% RSLogix 500 project O2 Sensor Calibration.RSS, saved by version 8.30.00.16 %
PROJECT "SIM_PLC"    % processor: Bul.1763 MicroLogix 1100 Series B %

PROGRAM FILES
  LAD 2 "MAIN"  4 rungs
  LAD 3 "IO"  5 rungs
  LAD 4 "CALIBRATE"  12 rungs
  LAD 5 "GAS VALVES"  3 rungs  % O2 Concentration Values to be read by O2 Sensor %

DATA FILES
  O0 OUTPUT  5 elements
  I1 INPUT  7 elements
  S2 STATUS  66 elements
  B3 BINARY  1 elements
  T4 TIMER  4 elements
  C5 COUNTER  1 elements
  R6 CONTROL  1 elements
  N7 INTEGER  14 elements
  F8 FLOAT  5 elements

LADDER 2 "MAIN"
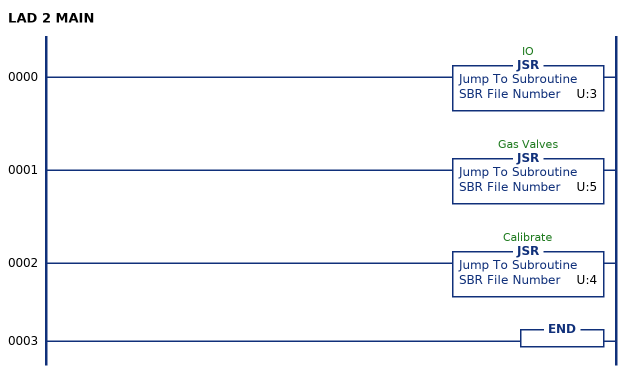
% Rung: 0 %
SOR JSR U:3 EOR
%   U:3  "IO" %
% Rung: 1 %
SOR JSR U:5 EOR
%   U:5  "Gas Valves" %
% Rung: 2 %
SOR JSR U:4 EOR
%   U:4  "Calibrate" %
% Rung: 3 %
SOR END EOR

LADDER 3 "IO"
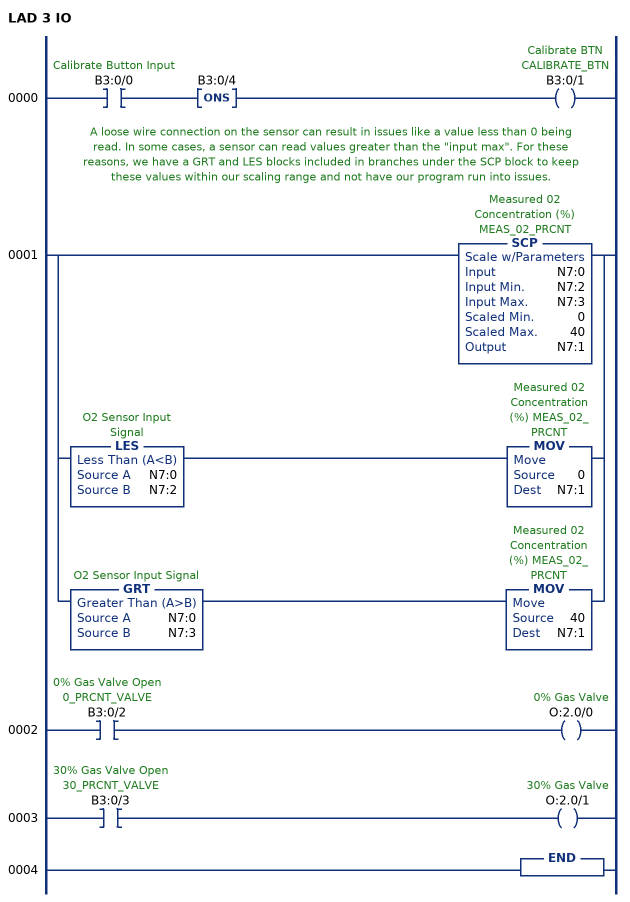
% Rung: 0 %
SOR XIC B3:0/0 ONS B3:0/4 OTE B3:0/1 EOR
%   B3:0/0  "Calibrate Button Input" %
%   B3:0/1  CALIBRATE_BTN  "Calibrate BTN" %
% Rung: 1 %
% A loose wire connection on the sensor can result in issues like a value less than 0 being read. In some cases, a sensor can read values greater than the "input max". For these reasons, we have a GRT and LES blocks included in branches under the SCP block to keep these values within our scaling range and not have our program run into issues. %
SOR BST SCP N7:0 N7:2 N7:3 0 40 N7:1 NXB LES N7:0 N7:2 MOV 0 N7:1 NXB GRT N7:0 N7:3 MOV 40 N7:1 BND EOR
%   N7:0  "O2 Sensor Input Signal" %
%   N7:2  "O2 Input Min" %
%   N7:3  "O2 Input Max" %
%   N7:1  MEAS_02_PRCNT  "Measured 02 Concentration (%)" %
% Rung: 2 %
SOR XIC B3:0/2 OTE O:2.0/0 EOR
%   B3:0/2  0_PRCNT_VALVE  "0% Gas Valve Open" %
%   O:2.0/0  "0% Gas Valve" %
% Rung: 3 %
SOR XIC B3:0/3 OTE O:2.0/1 EOR
%   B3:0/3  30_PRCNT_VALVE  "30% Gas Valve Open" %
%   O:2.0/1  "30% Gas Valve" %
% Rung: 4 %
SOR END EOR

LADDER 4 "CALIBRATE"
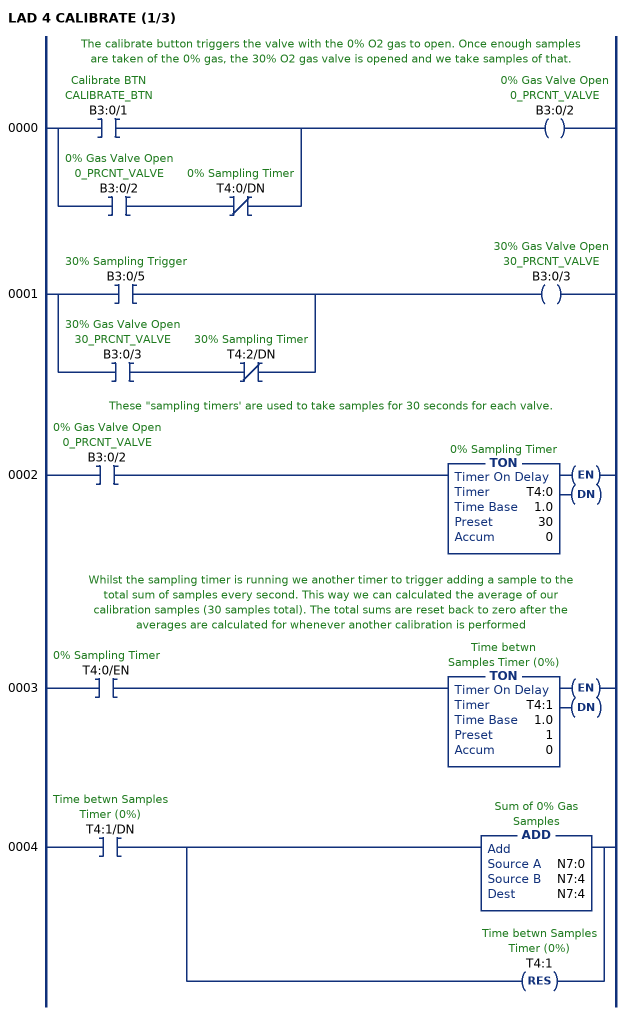
% Rung: 0 %
% The calibrate button triggers the valve with the 0% O2 gas to open. Once enough samples are taken of the 0% gas, the 30% O2 gas valve is opened and we take samples of that. %
SOR BST XIC B3:0/1 NXB XIC B3:0/2 XIO T4:0/DN BND OTE B3:0/2 EOR
%   B3:0/1  CALIBRATE_BTN  "Calibrate BTN" %
%   B3:0/2  0_PRCNT_VALVE  "0% Gas Valve Open" %
%   T4:0  "0% Sampling Timer" %
% Rung: 1 %
SOR BST XIC B3:0/5 NXB XIC B3:0/3 XIO T4:2/DN BND OTE B3:0/3 EOR
%   B3:0/5  "30% Sampling Trigger" %
%   B3:0/3  30_PRCNT_VALVE  "30% Gas Valve Open" %
%   T4:2  "30% Sampling Timer" %
% Rung: 2 %
% These "sampling timers' are used to take samples for 30 seconds for each valve. %
SOR XIC B3:0/2 TON T4:0 1.0 30 0 EOR
%   B3:0/2  0_PRCNT_VALVE  "0% Gas Valve Open" %
%   T4:0  "0% Sampling Timer" %
% Rung: 3 %
% Whilst the sampling timer is running we another timer to trigger adding a sample to the total sum of samples every second. This way we can calculated the average of our calibration samples (30 samples total). The total sums are reset back to zero after the averages are calculated for whenever another calibration is performed %
SOR XIC T4:0/EN TON T4:1 1.0 1 0 EOR
%   T4:0  "0% Sampling Timer" %
%   T4:1  "Time betwn Samples Timer (0%)" %
% Rung: 4 %
SOR XIC T4:1/DN BST ADD N7:0 N7:4 N7:4 NXB RES T4:1 BND EOR
%   T4:1  "Time betwn Samples Timer (0%)" %
%   N7:0  "O2 Sensor Input Signal" %
%   N7:4  "Sum of 0% Gas Samples" %

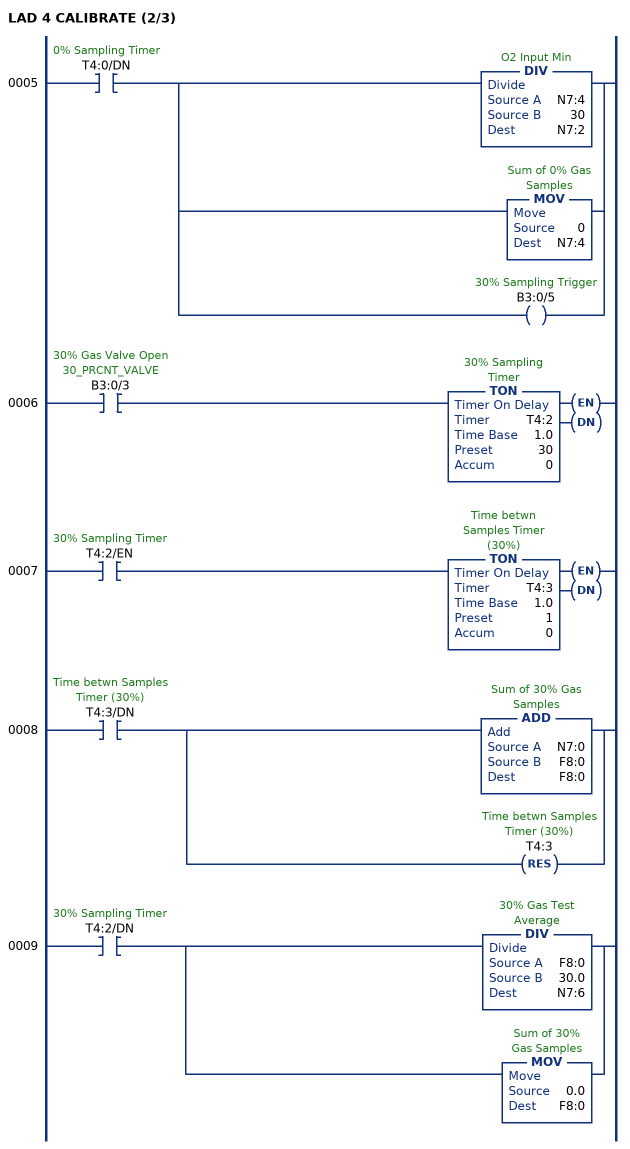
% Rung: 5 %
SOR XIC T4:0/DN BST DIV N7:4 30 N7:2 NXB MOV 0 N7:4 NXB OTE B3:0/5 BND EOR
%   T4:0  "0% Sampling Timer" %
%   N7:4  "Sum of 0% Gas Samples" %
%   N7:2  "O2 Input Min" %
%   B3:0/5  "30% Sampling Trigger" %
% Rung: 6 %
SOR XIC B3:0/3 TON T4:2 1.0 30 0 EOR
%   B3:0/3  30_PRCNT_VALVE  "30% Gas Valve Open" %
%   T4:2  "30% Sampling Timer" %
% Rung: 7 %
SOR XIC T4:2/EN TON T4:3 1.0 1 0 EOR
%   T4:2  "30% Sampling Timer" %
%   T4:3  "Time betwn Samples Timer (30%)" %
% Rung: 8 %
SOR XIC T4:3/DN BST ADD N7:0 F8:0 F8:0 NXB RES T4:3 BND EOR
%   T4:3  "Time betwn Samples Timer (30%)" %
%   N7:0  "O2 Sensor Input Signal" %
%   F8:0  "Sum of 30% Gas Samples" %
% Rung: 9 %
SOR XIC T4:2/DN BST DIV F8:0 30.0 N7:6 NXB MOV 0.0 F8:0 BND EOR
%   T4:2  "30% Sampling Timer" %
%   F8:0  "Sum of 30% Gas Samples" %
%   N7:6  "30% Gas Test Average" %

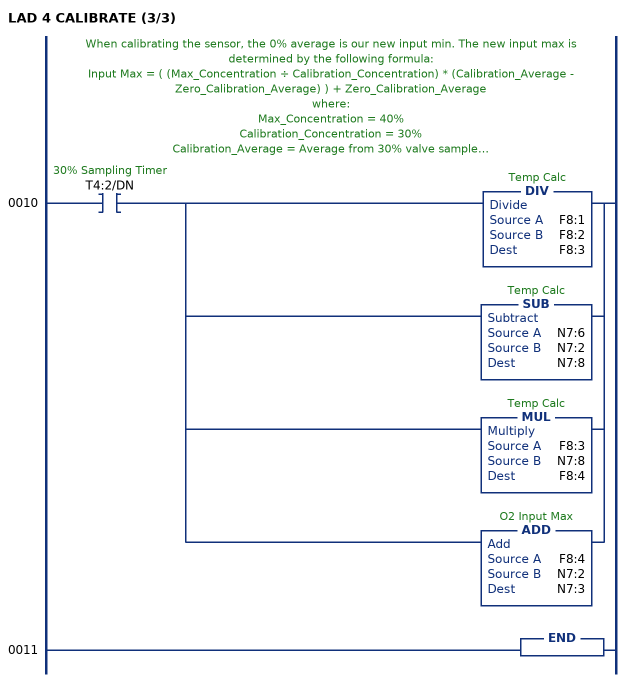
% Rung: 10 %
% When calibrating the sensor, the 0% average is our new input min. The new input max is determined by the following formula:
% 
% Input Max = ( (Max_Concentration ÷ Calibration_Concentration) * (Calibration_Average - Zero_Calibration_Average) ) + Zero_Calibration_Average
% 
% where:
% Max_Concentration = 40%
% Calibration_Concentration = 30%
% Calibration_Average = Average from 30% valve samples
% Zero_Calibration_Average = Average from 0% valve samples %
SOR XIC T4:2/DN BST DIV F8:1 F8:2 F8:3 NXB SUB N7:6 N7:2 N7:8 NXB MUL F8:3 N7:8 F8:4 NXB ADD F8:4 N7:2 N7:3 BND EOR
%   T4:2  "30% Sampling Timer" %
%   F8:1  "Max Concentration" %
%   F8:2  "Calibration Concentration" %
%   F8:3  "Temp Calc" %
%   N7:6  "30% Gas Test Average" %
%   N7:2  "O2 Input Min" %
%   N7:8  "Temp Calc" %
%   F8:4  "Temp Calc" %
%   N7:3  "O2 Input Max" %
% Rung: 11 %
SOR END EOR

LADDER 5 "GAS VALVES"    % O2 Concentration Values to be read by O2 Sensor %
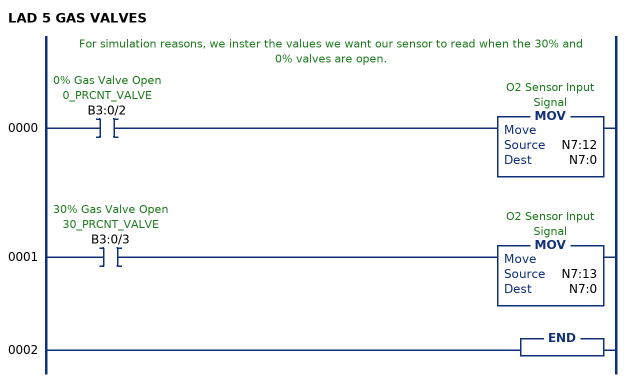
% Rung: 0 %
% For simulation reasons, we inster the values we want our sensor to read when the 30% and 0% valves are open. %
SOR XIC B3:0/2 MOV N7:12 N7:0 EOR
%   B3:0/2  0_PRCNT_VALVE  "0% Gas Valve Open" %
%   N7:12  "Custom 0% O2 Sensor Reading" %
%   N7:0  "O2 Sensor Input Signal" %
% Rung: 1 %
SOR XIC B3:0/3 MOV N7:13 N7:0 EOR
%   B3:0/3  30_PRCNT_VALVE  "30% Gas Valve Open" %
%   N7:13  "Custom 30% O2 Sensor Reading" %
%   N7:0  "O2 Sensor Input Signal" %
% Rung: 2 %
SOR END EOR

OTHER DOCUMENTED ADDRESSES
  PFILE:4  "Averaging of Calibra tion Samples"

DATA TABLE (non-zero values as saved)
DATA T4
% .PRE .ACC %
% T4:0 % 30 0
% T4:1 % 1 0
% T4:2 % 30 0
% T4:3 % 1 0
DATA N7
% N7:0 % 0 0 0 16383 0 0 0 0 0 0
% N7:10 % 0 0 100 11000
DATA F8
% F8:0 % 0 40 30 0 0
